SUBAPPLICATION Ventilsteuerung_Uebung_041 (* Lauflicht 8 mit einer Taste *)
  (* Standard: 61499-2 *)
  (* Version 1.0, 2023-10-23, franz *)
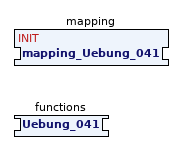
  SUBAPPS
    mapping : mapping_Uebung_041;
    functions : Uebung_041;
  END_SUBAPPS
END_SUBAPPLICATION
